(*
	RJM Maszyny sp. z o.o.
	autor 	: Rafał Osajda
	data	: 02.02.2024
	TC		: 3.1 4024.54
	wersja	: 0.0.1.0	: pełna obsługa

	Obsługa elektrozaworu do sterowania siłownikiem pneumatycznym.sterowanie 5 na 3 2 cewki zapowietrzone
*)
FUNCTION_BLOCK FB_Electrovalve_5on3_2Coil_Infected EXTENDS FB_Electrovalve

(*
	RJM Maszyny sp. z o.o.
	autor 	: Rafał Osajda
	data	: 21.02.2024
	TC		: 3.1 4024.54
	wersja	: 0.0.1.0	: pełna obsługa

	Ustawienie odpowiednich wyjść
*)
METHOD Contol : BOOL
VAR_INPUT
	eAction									: E_ElectrovalveAction;
END_VAR
CASE eAction OF
	E_ElectrovalveAction.e_EV_Out4_Deactive	:
		bCoilA								:= TRUE;
	E_ElectrovalveAction.e_EV_OUT4_Active	:
		bCoilA								:= FALSE;
	E_ElectrovalveAction.e_EV_Out2_Deactive	:
		bCoilB								:= TRUE;
	E_ElectrovalveAction.e_EV_Out2_Active	:
		bCoilB								:= FALSE;
	E_ElectrovalveAction.e_EV_ToStart	:
		bCoilA								:= TRUE;
		bCoilB								:= FALSE;
	E_ElectrovalveAction.e_EV_ToEnd		:
		bCoilA								:= FALSE;
		bCoilB								:= TRUE;
	E_ElectrovalveAction.e_EV_Stop		:
		bCoilA								:= FALSE;
		bCoilB								:= FALSE;
	E_ElectrovalveAction.e_EV_Reset			:
		bCoilA								:= FALSE;
		bCoilB								:= FALSE;
	E_ElectrovalveAction.e_EV_Active			:
		bCoilA								:= FALSE;
		bCoilB								:= FALSE;
	E_ElectrovalveAction.e_EV_Deactive		:
		bCoilA								:= FALSE;
		bCoilB								:= FALSE;	
END_CASE
END_METHOD

METHOD FB_init : BOOL
VAR_INPUT
	bInitRetains : BOOL; // if TRUE, the retain variables are initialized (warm start / cold start)
	bInCopyCode : BOOL;  // if TRUE, the instance afterwards gets moved into the copy code (online change)
END_VAR
THIS^.eType			:= E_ElectrovalveType.C2_5na3Z;
END_METHOD

END_FUNCTION_BLOCK

(* stored: Version 1.1.0.1
   POU FB_Electrovalve_5on3_2Coil_Infected: Id {f9a9052c-3bf3-09e5-23b0-206d47941a9f}, SpecialFunc None
   Method Contol: Id {b410a545-cfcd-05c3-03a5-9b6705863781}
   Method FB_init: Id {b99a4def-0aa6-4a9e-a1e5-5a26352a1c0e} *)
